{attribute 'linkalways'}
{attribute 'hide_all_locals'}
FUNCTION_BLOCK ValueWstringRead EXTENDS ValueBase IMPLEMENTS ValueRead
VAR
	thisValue : WSTRING(255);
END_VAR

{attribute 'call_after_global_init_slot' := '1'}
{attribute 'call_after_online_change_slot' := '1'}
METHOD PROTECTED GetThisAnyType
VAR_INPUT
END_VAR
thisAnyType := ToAnyType(thisValue);
END_METHOD

METHOD GetAsType : BOOL
VAR_INPUT
	destination : __SYSTEM.AnyType;
END_VAR
GetAsType := ConvertAnyType(thisAnyType, destination);
END_METHOD

METHOD GetAsString : T_MaxString
VAR_INPUT
END_VAR
GetAsString := WSTRING_TO_STRING(thisValue);
END_METHOD

METHOD Get : BOOL
VAR_INPUT
	destination : ANY;
END_VAR
Get := ConvertAnyType(thisAnyType, destination);
END_METHOD

METHOD FB_init : BOOL
VAR_INPUT
	bInitRetains : BOOL; // if TRUE, the retain variables are initialized (warm start / cold start)
	bInCopyCode : BOOL;  // if TRUE, the instance afterwards gets moved into the copy code (online change)
END_VAR
_ValueType := __SYSTEM.TYPE_CLASS.TYPE_WSTRING;
END_METHOD

{attribute 'monitoring' := 'call'}
PROPERTY Value : WSTRING(255)
GET
Value := thisValue;
END_GET
END_PROPERTY

END_FUNCTION_BLOCK

(* stored: Version 1.1.0.1
   POU ValueWstringRead: Id {076dc73c-b18e-4976-a455-e50151ece5f4}, SpecialFunc None
   Method GetThisAnyType: Id {bc33d865-8c5a-431b-8b29-9e93ddaed171}
   Method GetAsType: Id {420b0bc8-4195-4472-a8f0-bf92a9dd7c56}
   Method GetAsString: Id {ee0a8ad0-442d-49b0-8fd5-34ba692ba006}
   Method Get: Id {71e63da2-21df-48a3-947b-b88edce020a4}
   Method FB_init: Id {ee2d0e9c-d2c3-426f-8482-82667fa5fa6e}
   Property Value: Id {79215577-6aa4-4e51-8bda-1bf9da39a806}
   Get Get: Id {9c5d9086-b6f5-43af-bb5f-dda3c97ce727} *)
